// TIA Portal project "SimuMaqEmbalarAut" (V14)
// Simulação de uma maquina automatica para embalar produtos

(* hardware
DEVICE "S7-1200 station_1"  S7-1200 Station
   slot 0: "Rack_0"  S7-1200 Rack  Rack  V1.0
   slot 1: "Embaladora automatica"  CPU 1214C DC/DC/DC  6ES7 214-1AG40-0XB0  V4.2
*)

// ===== PLC "Embaladora automatica"  CPU 1214C DC/DC/DC =====

VAR_GLOBAL   // PLC tag table "Default tag table"
   ""SensorProduto"" AT %I0.0 : Bool;
   ""SensorCaixa"" AT %I0.1 : Bool;
   ""ChaveOnOff"" AT %I0.2 : Bool;
   ""MotorEsteiraCaixa"" AT %Q0.0 : Bool;
   ""MotorEsteiraProduto"" AT %Q0.1 : Bool;
   ""LuzVerde"" AT %Q0.2 : Bool;
   ""LuzAmarela"" AT %Q0.3 : Bool;
   ""LuzVermelha"" AT %Q0.4 : Bool;
END_VAR